// TIA Portal V20 export
DATA_BLOCK "PM5"   // DB279
// stored: MemoryReserve 100
   VAR
      "SIDE TAPE CUTTER FORWARD" : Bool;
      "SIDE TAPE CUTTER BACKWARD" : Bool;
      "SIDE TAPE CUTTER CLAMP FORWARD" : Bool;
      "SIDE TAPE CUTTER CLAMP BACKWARD" : Bool;
      "SIDE TAPE CLAMP CLOSE" : Bool;
      "SIDE TAPE CLAMP OPEN" : Bool;
      "SIDE TAPE TENSION FORWARD" : Bool;
      "SIDE TAPE TENSION BACKWARD" : Bool;
      "SIDE TAPE LOADING FORWARD" : Bool;
      "SIDE TAPE LOADING BACKWARD" : Bool;
      SPARE : Bool;
      SPARE_1 : Bool;
      SPARE_2 : Bool;
      SPARE_3 : Bool;
      SPARE_4 : Bool;
      SPARE_5 : Bool;
   END_VAR
BEGIN
END_DATA_BLOCK
